{attribute addProperty BoxType "CU1123-0010-0016"}
{attribute addProperty Id "A_0003_CU1124_0000_0016A_0003_CU1124_0000_0016_F6CF179A950118.75"}
{attribute addProperty CRC "3245134003"}
{attribute addProperty SizeInBites "950"}
{attribute addProperty SizeInBytes "118.75"}
TYPE A_0002_CU1123_0010_0016_C16CD0B3 EXTENDS CU1123_179A0949 :
STRUCT
	{attribute addProperty Name "A_0003_CU1124_0000_0016"}
	A_0003_CU1124_0000_0016 : A_0003_CU1124_0000_0016_F6CF179A;
END_STRUCT
END_TYPE

(* stored: Version 1.2.0.0, ProductVersion 3.1.4024.9
   DUT A_0002_CU1123_0010_0016_C16CD0B3: Id {73eec53a-ae4d-4d5e-a4d6-9e4c0a0f3781} *)
